PROGRAM DoorFaults
VAR
	header_left : ARRAY [1..5] OF WORD := [16#2A2A, 16#2A2A, 16#2A44, 16#4F4F, 16#5220];
	header_right: ARRAY [1..5] OF WORD := [16#4641, 16#554C, 16#542A, 16#2A2A, 16#2A2A];
	
	usr_ok: ARRAY [1..5] OF WORD := [16#2055, 16#5352, 16#204F, 16#4B20, 16#2020];
	usr_fault: ARRAY [1..5] OF WORD := [16#2055, 16#5352, 16#2046, 16#4C54, 16#2020];
	                                   
	usl_ok: ARRAY [1..5] OF WORD := [16#2055, 16#534C, 16#204F, 16#4B20, 16#2020];
	usl_fault: ARRAY [1..5] OF WORD := [16#2055, 16#534C, 16#2046, 16#4C54, 16#2020];
	                                   
	dsr_ok: ARRAY [1..5] OF WORD := [16#2044, 16#5352, 16#204F, 16#4B20, 16#2020];
	dsr_fault: ARRAY [1..5] OF WORD := [16#2044, 16#5352, 16#2046, 16#4C54, 16#2020];
	                                   
	dsl_ok: ARRAY [1..5] OF WORD := [16#2044, 16#534C, 16#204F, 16#4B20, 16#2020];
	dsl_fault: ARRAY [1..5] OF WORD := [16#2044, 16#534C, 16#2046, 16#4C54, 16#2020];
	
	
	tick: INT := 0;
END_VAR

GV_MODBUS.oneLeft:= header_left;
GV_MODBUS.oneRight:= header_right;

GV_MODBUS.twoLeft:= GV_MODBUS.blank;
GV_MODBUS.twoRight:= GV_MODBUS.blank;

IF GV_LIFT.DOOR_1_INDICATOR_OUT THEN
	GV_MODBUS.threeLeft:= dsl_fault;
ELSE
	GV_MODBUS.threeLeft:= dsl_ok;
END_IF  

IF GV_LIFT.DOOR_2_INDICATOR_OUT THEN
	GV_MODBUS.threeRight:= dsr_fault;
ELSE
	GV_MODBUS.threeRight:= dsr_ok;
END_IF

IF GV_LIFT.DOOR_3_INDICATOR_OUT THEN
	GV_MODBUS.fourLeft:= usl_fault;
ELSE
	GV_MODBUS.fourLeft:= usl_ok;
END_IF

IF GV_LIFT.DOOR_4_INDICATOR_OUT THEN
	GV_MODBUS.fourRight:= usr_fault;
ELSE
	GV_MODBUS.fourRight:= usr_ok;
END_IF


IF tick >= GV_MODBUS.refreshInterval THEN
	Execute_Write_Screen();
	tick := 0;
END_IF

tick := tick + 1;

END_PROGRAM

(* stored: Version 1.1.0.1, ProductVersion 3.1.4022.12
   POU DoorFaults: Id {17bb635c-b6f7-4157-a8d6-2a30cc4dea9b}, SpecialFunc None *)
